TYPE ST_DCSwitchgear_Get :
STRUCT
	b_CouplingState					: BOOL;
	r_Current						: REAL;
	r_Power							: REAL;
	r_Voltage						: REAL;
	r_RatedCurrent					: REAL;
END_STRUCT
END_TYPE

(* stored: Version 1.1.0.1, ProductVersion 3.1.4024.12
   DUT ST_DCSwitchgear_Get: Id {1eee37a2-3d57-4cc4-8f20-af24b3850966} *)
